FUNCTION iGetNextBufferPointer : INT
VAR_INPUT
	iBufferSize : INT;
	iActualPointerValue : INT;
END_VAR
VAR
	retVal : INT;
END_VAR

retVal := iActualPointerValue + 1;
IF retVal >= iBufferSize THEN retVal := 0; END_IF;
iGetNextBufferPointer := retVal;

END_FUNCTION

(* stored: Version 1.1.0.1, ProductVersion 3.1.4024.12
   POU iGetNextBufferPointer: Id {c4b40ba6-e249-4b6c-bc0d-9b679ded4000}, SpecialFunc None *)
